{attribute 'qualified_only'}
VAR_GLOBAL CONSTANT
	ENTITY_CAP		: UDINT(1..16#7FFFFFFF) := 20;
	COMP_CAP		: UDINT(1..16#7FFFFFFF) := 100;
	
	DEBUGMSG_CAP	: UDINT(1..16#7FFFFFFF) := 10;
	DEBUGSTR_CAP	: UDINT(1..16#7FFFFFFF) := 500;
	
	SIGNAL_CAP		: UDINT(1..16#7FFFFFFF) := 20;
	RECEIVER_CAP	: UDINT(1..16#7FFFFFFF) := 100;
END_VAR

(* stored: Version 1.1.0.1
   GVL Param: Id {bc9b684f-96ba-4011-afc3-650f65d44b69}, ParameterList True *)
